// TIA Portal V20 program export: 4 tag tables, 3 data types, 2 data blocks, 7 code blocks (in call order from the OBs), 2 instance data blocks

VAR_GLOBAL   // PLC tag table "Inputs Equipment"
   i_xSabload_Part1_p1_LR AT %I1.0 : Bool;   // Input - Sabload part 1 sensor - table P1 for Left and Right Jig
   i_xSabload_Part2_p1_L AT %I1.1 : Bool;   // Input - Sabload part 2 sensor - table P1 for Left Jig
   i_xSabload_Part3_p1_L AT %I1.2 : Bool;   // Input - Sabload part 3 sensor - table P1 for Left Jig
   i_xSabload_Part4_p1_LR AT %I1.3 : Bool;   // Input - Sabload part 4 sensor - table P1 for Left and Right Jig
   i_xSabload_Part2_p1_R AT %I1.4 : Bool;   // Input - Sabload part 2 sensor - table P1 for Right Jig
   i_xSabload_Part3_p1_R AT %I1.5 : Bool;   // Input - Sabload part 3 sensor - table P1 for Right Jig
   i_xSabload_Part1_p2_LR AT %I1.6 : Bool;   // Input - Sabload part 1 sensor - table P2 for Left and Right Jig
   i_xSabload_Part2_p2_L AT %I1.7 : Bool;   // Input - Sabload part 2 sensor - table P2 for Left Jig
   i_xSabload_Part3_p2_L AT %I2.0 : Bool;   // Input - Sabload part 3 sensor - table P2 for Left Jig
   i_xSabload_Part4_p2_LR AT %I2.1 : Bool;   // Input - Sabload part 4 sensor - table P2 for Left and Right Jig
   i_xSabload_Part2_p2_R AT %I2.2 : Bool;   // Input - Sabload part 2 sensor - table P2 for Right Jig
   i_xSabload_Part3_p2_R AT %I2.3 : Bool;   // Input - Sabload part 3 sensor - table P2 for Right Jig
   i_xBas342_ProgBit0 AT %I0.0 : Bool;   // Input - Bas 342 prog bit 0 for left side Jig
   i_xBas342_ProgBit1 AT %I0.1 : Bool;   // Input - Bas 342 prog bit 1 for Right side Jig
   i_xTableCheck_JigPresent_p1 AT %I0.2 : Bool;   // Input: TableCheck process 1 Sensor for Jig presence for Table P1
   i_xTableCheck_JigPresent_p2 AT %I0.3 : Bool;   // Input: TableCheck process 1 Sensor for Jig presence for Table P2
END_VAR

VAR_GLOBAL   // PLC tag table "OutPut Equipment"
   q_xTableCheck_LampNG_p1 AT %Q5.0 : Bool;   // Output - indication lamp, NO good operation for table P1
   q_xTableCheck_LampOK_p1 AT %Q5.1 : Bool;   // Output - indication lamp, Ok operation for table P1
   q_xTableCheck_LampNG_p2 AT %Q5.2 : Bool;   // Output - indication lamp, NO good operation for table P2
   q_xTableCheck_LampOK_p2 AT %Q5.3 : Bool;   // Output - indication lamp, Ok operation for table P2
END_VAR

VAR_GLOBAL   // PLC tag table "Inputs Machine"
END_VAR

VAR_GLOBAL   // PLC tag table "Output Machine"
END_VAR

TYPE "UDT-BAS342"
VERSION : 0.1
   STRUCT
      Sts : Struct   // Status structure
         xFaulted : Bool;   // wrong program
         xWrongJigProgram : Bool;   // Wrong jig Program by the bus machine
         xNoprogram : Bool;
      END_STRUCT;
      Cmd : Struct   // Command structure
         xCorrectJigProgram : Bool;   // Correct jig Program by the bus machine
         xLeftJig : Bool;   // Bit for the program form the Bas machine
         xRightJig : Bool;   // Bit for the program form the Bas machine
         Spare : Bool;
      END_STRUCT;
      Cfg : Struct   // Configuration structure
         xSpare : Bool;   // Spare
      END_STRUCT;
      Flt : Struct   // Fault structure
         wTrigger : Word;   // Fault triggers
      END_STRUCT;
   END_STRUCT;

END_TYPE

TYPE "UDT-SABload"
VERSION : 0.1
   STRUCT
      Sts : Struct   // Status structure
         axSesnor : Array[1..4] of Bool;
         xCorrectpart : Bool;   // correct part indicaton
         faulted : Bool;   // the module is faulted
         State : Int;   // state machine value
      END_STRUCT;
      Cmd : Struct   // Command structure
         spare : Bool;
      END_STRUCT;
      Cfg : Struct   // Configuration structure
         xSpare : Bool;   // Spare
      END_STRUCT;
      Flt : Struct   // Fault structure
         wTrigger : Word;   // Fault triggers
      END_STRUCT;
   END_STRUCT;

END_TYPE

TYPE "UDT-TableCheck"
VERSION : 0.1
   STRUCT
      Sts : Struct   // Status structure
         xFaulted : Bool;   // System is in faulted state
         xStartSensor : Bool;   // Spare
         xLeftJigplaced : Bool;   // Left Jig is pleased with Left Bas sew program 
         xRightJigPlaced : Bool;   // Right Jig is pleased with Right Bas sew program 
         "xCorrect part" : Bool;   //  the part of the airbage is placed correctly
      END_STRUCT;
      Cmd : Struct   // Command structure
         xJigpresent : Bool;
         spare : Bool;
      END_STRUCT;
      Flt : Struct   // fault structure
         wTrigger : Byte;   // fault trigger word
      END_STRUCT;
   END_STRUCT;

END_TYPE

DATA_BLOCK "DB - Equipment"   // DB4
{ S7_Optimized_Access := 'TRUE' }
// stored: MemoryReserve 100
   VAR
      TableCheckProcess1 : "UDT-TableCheck";
      TableCheckProcess2 : "UDT-TableCheck";
      "SabLaodProcess1-L" { S7_SetPoint := 'True'} : "UDT-SABload";
      "SabLaodProcess1-R" { S7_SetPoint := 'True'} : "UDT-SABload";
      "SabLaodProcess2-L" { S7_SetPoint := 'True'} : "UDT-SABload";
      "SabLaodProcess2-R" { S7_SetPoint := 'True'} : "UDT-SABload";
      Bas342 { S7_SetPoint := 'True'} : "UDT-BAS342";
   END_VAR
BEGIN
END_DATA_BLOCK

DATA_BLOCK "DB - Machine"   // DB3
{ S7_Optimized_Access := 'TRUE' }
// stored: MemoryReserve 100
BEGIN
END_DATA_BLOCK

ORGANIZATION_BLOCK "Main"   // OB1, LAD, ProgramCycle
TITLE = "Main Program Sweep (Cycle)"
{ S7_Optimized_Access := 'TRUE' }
// stored: SetENOAutomatically false
   VAR_INPUT
      Initial_Call : Bool;   // Initial call of this OB
      Remanence : Bool;   // =True, if remanent data are available
   END_VAR
BEGIN

REGION Network 1: CALL - Main machine modules (Not used)
   // Call of the application's main machine functions (NOT used)
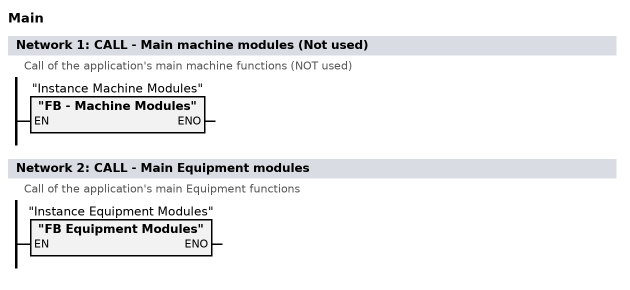
   RUNG wire#powerrail
      "Instance Machine Modules"()
   END_RUNG
   // the same network as SCL:
   "Instance Machine Modules"();   // "FB - Machine Modules"
END_REGION

REGION Network 2: CALL - Main Equipment modules
   // Call of the application's main Equipment functions
   RUNG wire#powerrail
      "Instance Equipment Modules"()
   END_RUNG
   // the same network as SCL:
   "Instance Equipment Modules"();   // "FB Equipment Modules"
END_REGION
END_ORGANIZATION_BLOCK

FUNCTION_BLOCK "FB - Machine Modules"   // FB1, LAD
TITLE = Machine - Modules
{ S7_Optimized_Access := 'TRUE' }
// stored: MemoryReserve 100, SetENOAutomatically false
BEGIN

REGION Network 1: StateHandler process 1 - table
END_REGION

REGION Network 2: StateHandler process 2 - table
END_REGION
END_FUNCTION_BLOCK

FUNCTION_BLOCK "FB Equipment Modules"   // FB2, LAD
TITLE = FB - Equipment Modules
{ S7_Optimized_Access := 'TRUE' }
// stored: MemoryReserve 100, SetENOAutomatically false
   VAR
      "Instance - Bas342" { S7_SetPoint := 'True'} : "FB - Bas342";
      "Instance - TableCheck - Process1" { S7_SetPoint := 'True'} : "FB - TableCheck";
      "Instance - TableCheck - Process2" { S7_SetPoint := 'True'} : "FB - TableCheck";
      "Instance - Sabload - P1 Left" { S7_SetPoint := 'True'} : "FB - Sabload";
      "Instance - Sabload - P1 Right" { S7_SetPoint := 'True'} : "FB - Sabload";
      "Instance - Sabload - P2 Left" { S7_SetPoint := 'True'} : "FB - Sabload";
      "Instance - Sabload - P2 Right" { S7_SetPoint := 'True'} : "FB - Sabload";
   END_VAR
BEGIN

REGION Network 1: Module - Bas342
   // Call of the Bas342 module.
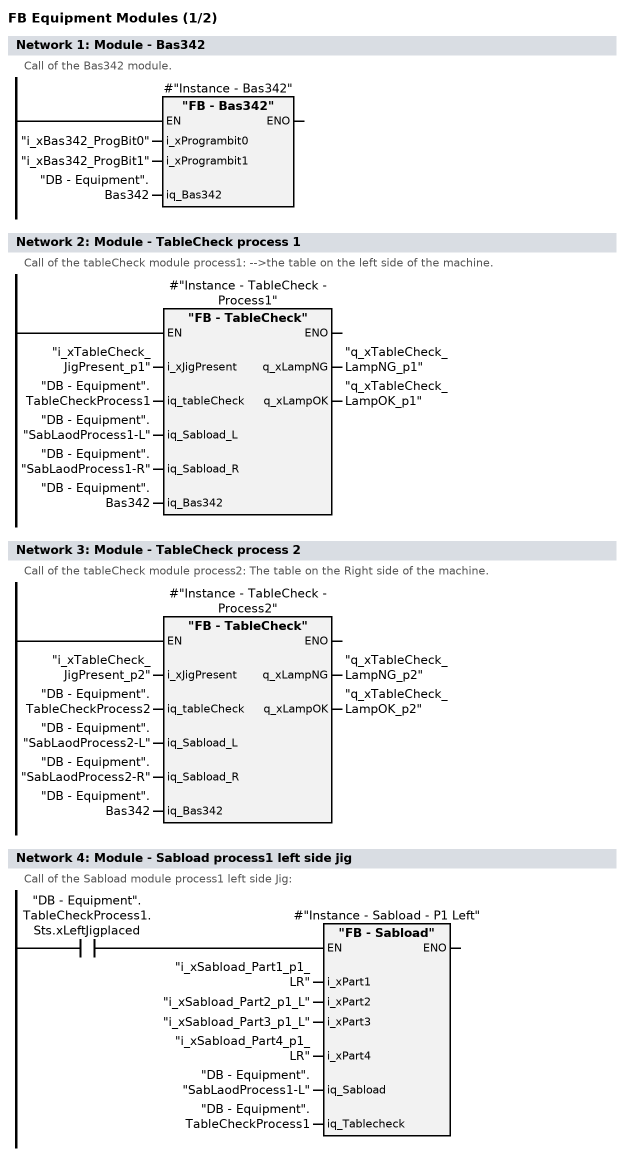
   RUNG wire#powerrail
      #"Instance - Bas342"(i_xProgrambit0 := "i_xBas342_ProgBit0", i_xProgrambit1 := "i_xBas342_ProgBit1", iq_Bas342 := "DB - Equipment".Bas342)
   END_RUNG
   // the same network as SCL:
   #"Instance - Bas342"(i_xProgrambit0 := "i_xBas342_ProgBit0",   // "FB - Bas342"
                        i_xProgrambit1 := "i_xBas342_ProgBit1",
                        iq_Bas342 := "DB - Equipment".Bas342);
END_REGION

REGION Network 2: Module - TableCheck process 1
   // Call of the tableCheck module process1: -->the table on the left side of the machine.
   RUNG wire#powerrail
      #"Instance - TableCheck - Process1"(i_xJigPresent := "i_xTableCheck_JigPresent_p1", iq_tableCheck := "DB - Equipment".TableCheckProcess1, iq_Sabload_L := "DB - Equipment"."SabLaodProcess1-L", iq_Sabload_R := "DB - Equipment"."SabLaodProcess1-R", iq_Bas342 := "DB - Equipment".Bas342, q_xLampNG => "q_xTableCheck_LampNG_p1", q_xLampOK => "q_xTableCheck_LampOK_p1")
   END_RUNG
   // the same network as SCL:
   #"Instance - TableCheck - Process1"(i_xJigPresent := "i_xTableCheck_JigPresent_p1",   // "FB - TableCheck"
                           iq_tableCheck := "DB - Equipment".TableCheckProcess1,
                           iq_Sabload_L := "DB - Equipment"."SabLaodProcess1-L",
                           iq_Sabload_R := "DB - Equipment"."SabLaodProcess1-R",
                           iq_Bas342 := "DB - Equipment".Bas342,
                           q_xLampNG => "q_xTableCheck_LampNG_p1",
                           q_xLampOK => "q_xTableCheck_LampOK_p1");
END_REGION

REGION Network 3: Module - TableCheck process 2
   // Call of the tableCheck module process2: The table on the Right side of the machine.
   RUNG wire#powerrail
      #"Instance - TableCheck - Process2"(i_xJigPresent := "i_xTableCheck_JigPresent_p2", iq_tableCheck := "DB - Equipment".TableCheckProcess2, iq_Sabload_L := "DB - Equipment"."SabLaodProcess2-L", iq_Sabload_R := "DB - Equipment"."SabLaodProcess2-R", iq_Bas342 := "DB - Equipment".Bas342, q_xLampNG => "q_xTableCheck_LampNG_p2", q_xLampOK => "q_xTableCheck_LampOK_p2")
   END_RUNG
   // the same network as SCL:
   #"Instance - TableCheck - Process2"(i_xJigPresent := "i_xTableCheck_JigPresent_p2",   // "FB - TableCheck"
                           iq_tableCheck := "DB - Equipment".TableCheckProcess2,
                           iq_Sabload_L := "DB - Equipment"."SabLaodProcess2-L",
                           iq_Sabload_R := "DB - Equipment"."SabLaodProcess2-R",
                           iq_Bas342 := "DB - Equipment".Bas342,
                           q_xLampNG => "q_xTableCheck_LampNG_p2",
                           q_xLampOK => "q_xTableCheck_LampOK_p2");
END_REGION

REGION Network 4: Module - Sabload process1 left side jig
   // Call of the Sabload module process1 left side Jig:
   RUNG wire#powerrail
      Contact( "DB - Equipment".TableCheckProcess1.Sts.xLeftJigplaced )
      #"Instance - Sabload - P1 Left"(i_xPart1 := "i_xSabload_Part1_p1_LR", i_xPart2 := "i_xSabload_Part2_p1_L", i_xPart3 := "i_xSabload_Part3_p1_L", i_xPart4 := "i_xSabload_Part4_p1_LR", iq_Sabload := "DB - Equipment"."SabLaodProcess1-L", iq_Tablecheck := "DB - Equipment".TableCheckProcess1)
   END_RUNG
   // the same network as SCL:
   IF "DB - Equipment".TableCheckProcess1.Sts.xLeftJigplaced THEN
       #"Instance - Sabload - P1 Left"(i_xPart1 := "i_xSabload_Part1_p1_LR",   // "FB - Sabload"
                               i_xPart2 := "i_xSabload_Part2_p1_L",
                               i_xPart3 := "i_xSabload_Part3_p1_L",
                               i_xPart4 := "i_xSabload_Part4_p1_LR",
                               iq_Sabload := "DB - Equipment"."SabLaodProcess1-L",
                               iq_Tablecheck := "DB - Equipment".TableCheckProcess1);
   END_IF;
END_REGION

REGION Network 5: Module - Sabload process1 Right side jig
   // Call of the Sabload module process1 Right side Jig:
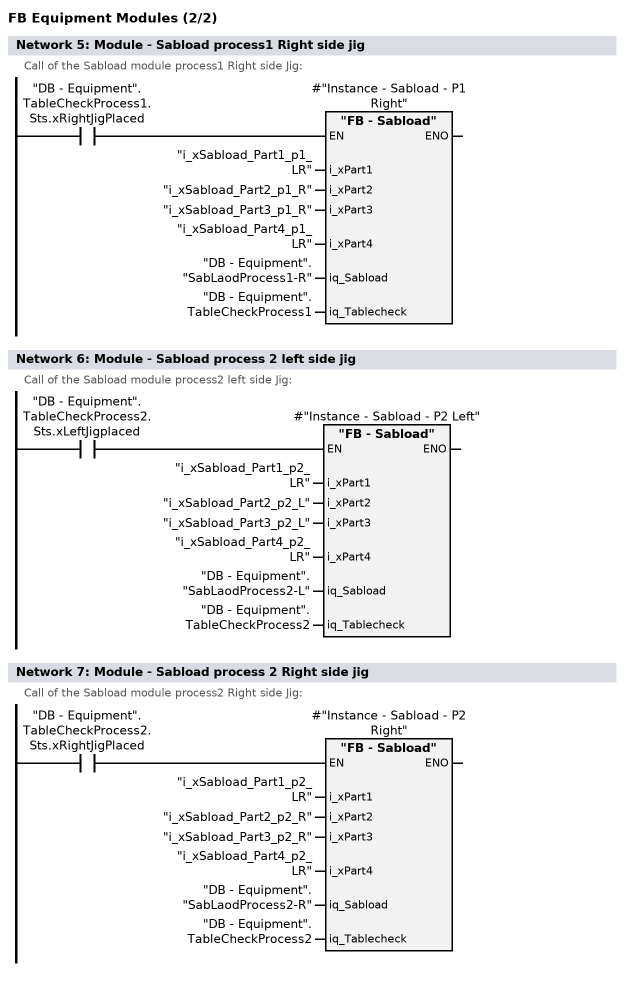
   RUNG wire#powerrail
      Contact( "DB - Equipment".TableCheckProcess1.Sts.xRightJigPlaced )
      #"Instance - Sabload - P1 Right"(i_xPart1 := "i_xSabload_Part1_p1_LR", i_xPart2 := "i_xSabload_Part2_p1_R", i_xPart3 := "i_xSabload_Part3_p1_R", i_xPart4 := "i_xSabload_Part4_p1_LR", iq_Sabload := "DB - Equipment"."SabLaodProcess1-R", iq_Tablecheck := "DB - Equipment".TableCheckProcess1)
   END_RUNG
   // the same network as SCL:
   IF "DB - Equipment".TableCheckProcess1.Sts.xRightJigPlaced THEN
       #"Instance - Sabload - P1 Right"(i_xPart1 := "i_xSabload_Part1_p1_LR",   // "FB - Sabload"
                               i_xPart2 := "i_xSabload_Part2_p1_R",
                               i_xPart3 := "i_xSabload_Part3_p1_R",
                               i_xPart4 := "i_xSabload_Part4_p1_LR",
                               iq_Sabload := "DB - Equipment"."SabLaodProcess1-R",
                               iq_Tablecheck := "DB - Equipment".TableCheckProcess1);
   END_IF;
END_REGION

REGION Network 6: Module - Sabload process 2 left side jig
   // Call of the Sabload module process2 left side Jig:
   RUNG wire#powerrail
      Contact( "DB - Equipment".TableCheckProcess2.Sts.xLeftJigplaced )
      #"Instance - Sabload - P2 Left"(i_xPart1 := "i_xSabload_Part1_p2_LR", i_xPart2 := "i_xSabload_Part2_p2_L", i_xPart3 := "i_xSabload_Part3_p2_L", i_xPart4 := "i_xSabload_Part4_p2_LR", iq_Sabload := "DB - Equipment"."SabLaodProcess2-L", iq_Tablecheck := "DB - Equipment".TableCheckProcess2)
   END_RUNG
   // the same network as SCL:
   IF "DB - Equipment".TableCheckProcess2.Sts.xLeftJigplaced THEN
       #"Instance - Sabload - P2 Left"(i_xPart1 := "i_xSabload_Part1_p2_LR",   // "FB - Sabload"
                               i_xPart2 := "i_xSabload_Part2_p2_L",
                               i_xPart3 := "i_xSabload_Part3_p2_L",
                               i_xPart4 := "i_xSabload_Part4_p2_LR",
                               iq_Sabload := "DB - Equipment"."SabLaodProcess2-L",
                               iq_Tablecheck := "DB - Equipment".TableCheckProcess2);
   END_IF;
END_REGION

REGION Network 7: Module - Sabload process 2 Right side jig
   // Call of the Sabload module process2 Right side Jig:
   RUNG wire#powerrail
      Contact( "DB - Equipment".TableCheckProcess2.Sts.xRightJigPlaced )
      #"Instance - Sabload - P2 Right"(i_xPart1 := "i_xSabload_Part1_p2_LR", i_xPart2 := "i_xSabload_Part2_p2_R", i_xPart3 := "i_xSabload_Part3_p2_R", i_xPart4 := "i_xSabload_Part4_p2_LR", iq_Sabload := "DB - Equipment"."SabLaodProcess2-R", iq_Tablecheck := "DB - Equipment".TableCheckProcess2)
   END_RUNG
   // the same network as SCL:
   IF "DB - Equipment".TableCheckProcess2.Sts.xRightJigPlaced THEN
       #"Instance - Sabload - P2 Right"(i_xPart1 := "i_xSabload_Part1_p2_LR",   // "FB - Sabload"
                               i_xPart2 := "i_xSabload_Part2_p2_R",
                               i_xPart3 := "i_xSabload_Part3_p2_R",
                               i_xPart4 := "i_xSabload_Part4_p2_LR",
                               iq_Sabload := "DB - Equipment"."SabLaodProcess2-R",
                               iq_Tablecheck := "DB - Equipment".TableCheckProcess2);
   END_IF;
END_REGION
END_FUNCTION_BLOCK

FUNCTION_BLOCK "FB - Bas342"   // FB6, LAD
TITLE = Equipment - Bas342
{ S7_Optimized_Access := 'TRUE' }
// This Function blick contain all the logic for controlling a Bas342 module.
// --This module basically for BAS342 sewing machine.
// It is consist of two program bits from BAS342.
// >> Block created by: Engr. Awais Ali
// >> Block creation date:  08-10-2025
// stored: MemoryReserve 100, SetENOAutomatically false
   VAR_INPUT
      i_xProgrambit0 : Bool;
      i_xProgrambit1 : Bool;
   END_VAR
   VAR_IN_OUT
      iq_Bas342 : "UDT-BAS342";
   END_VAR
BEGIN

REGION Network 1: Control - left jig
   // Bit 0 represent the left jig program.
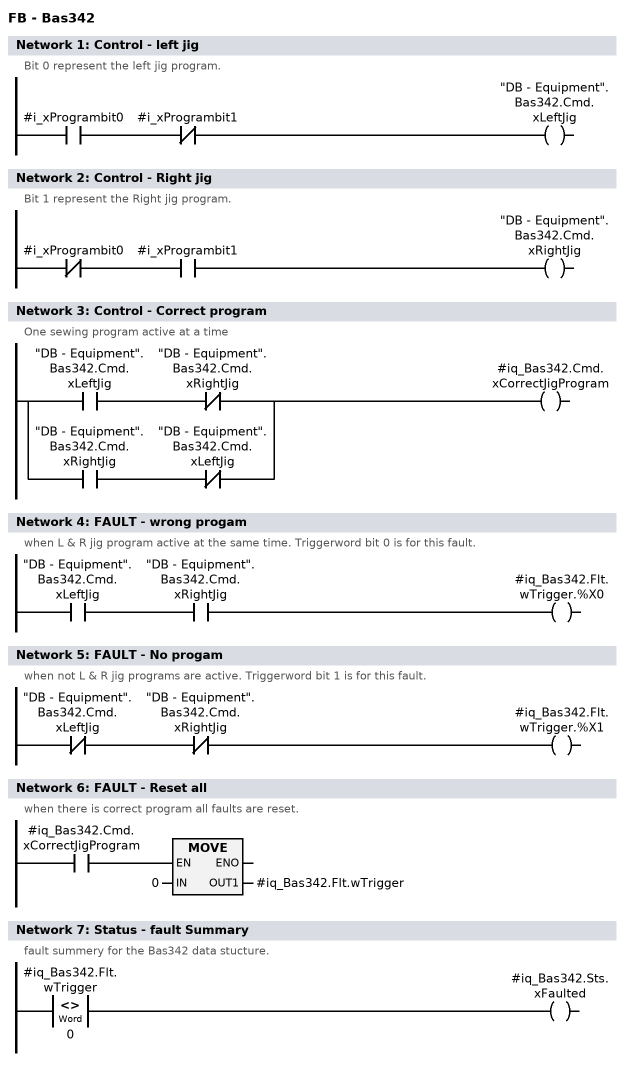
   RUNG wire#powerrail
      Contact( #i_xProgrambit0 )
      I_Contact( #i_xProgrambit1 )
      Coil( "DB - Equipment".Bas342.Cmd.xLeftJig )
   END_RUNG
   // the same network as SCL:
   "DB - Equipment".Bas342.Cmd.xLeftJig := #i_xProgrambit0 AND NOT #i_xProgrambit1;
END_REGION

REGION Network 2: Control - Right jig
   // Bit 1 represent the Right jig program.
   RUNG wire#powerrail
      I_Contact( #i_xProgrambit0 )
      Contact( #i_xProgrambit1 )
      Coil( "DB - Equipment".Bas342.Cmd.xRightJig )
   END_RUNG
   // the same network as SCL:
   "DB - Equipment".Bas342.Cmd.xRightJig := NOT #i_xProgrambit0 AND #i_xProgrambit1;
END_REGION

REGION Network 3: Control - Correct program
   // One sewing program active at a time
   RUNG wire#powerrail
      Contact( "DB - Equipment".Bas342.Cmd.xLeftJig )
      I_Contact( "DB - Equipment".Bas342.Cmd.xRightJig )
      wire#w1
      Coil( #iq_Bas342.Cmd.xCorrectJigProgram )
   END_RUNG
   RUNG wire#powerrail
      Contact( "DB - Equipment".Bas342.Cmd.xRightJig )
      I_Contact( "DB - Equipment".Bas342.Cmd.xLeftJig )
   END_RUNG wire#w1
   // the same network as SCL:
   #iq_Bas342.Cmd.xCorrectJigProgram := ("DB - Equipment".Bas342.Cmd.xLeftJig AND NOT "DB - Equipment".Bas342.Cmd.xRightJig) OR ("DB - Equipment".Bas342.Cmd.xRightJig AND NOT "DB - Equipment".Bas342.Cmd.xLeftJig);
END_REGION

REGION Network 4: FAULT - wrong progam
   // when L & R jig program active at the same time. Triggerword bit 0 is for this fault.
   RUNG wire#powerrail
      Contact( "DB - Equipment".Bas342.Cmd.xLeftJig )
      Contact( "DB - Equipment".Bas342.Cmd.xRightJig )
      Coil( #iq_Bas342.Flt.wTrigger.%X0 )
   END_RUNG
   // the same network as SCL:
   #iq_Bas342.Flt.wTrigger.%X0 := "DB - Equipment".Bas342.Cmd.xLeftJig AND "DB - Equipment".Bas342.Cmd.xRightJig;
END_REGION

REGION Network 5: FAULT - No progam
   // when not L & R jig programs are active. Triggerword bit 1 is for this fault.
   RUNG wire#powerrail
      I_Contact( "DB - Equipment".Bas342.Cmd.xLeftJig )
      I_Contact( "DB - Equipment".Bas342.Cmd.xRightJig )
      Coil( #iq_Bas342.Flt.wTrigger.%X1 )
   END_RUNG
   // the same network as SCL:
   #iq_Bas342.Flt.wTrigger.%X1 := NOT "DB - Equipment".Bas342.Cmd.xLeftJig AND NOT "DB - Equipment".Bas342.Cmd.xRightJig;
END_REGION

REGION Network 6: FAULT - Reset all
   // when there is correct program all faults are reset.
   RUNG wire#powerrail
      Contact( #iq_Bas342.Cmd.xCorrectJigProgram )
      Move(in := 0, out1 => #iq_Bas342.Flt.wTrigger)
   END_RUNG
   // the same network as SCL:
   IF #iq_Bas342.Cmd.xCorrectJigProgram THEN #iq_Bas342.Flt.wTrigger := 0; END_IF;
END_REGION

REGION Network 7: Status - fault Summary
   // fault summery for the Bas342 data stucture.
   RUNG wire#powerrail
      { S7_Templates := "SrcType := Word" } NE_Contact(in1 := #iq_Bas342.Flt.wTrigger, in2 := 0)
      Coil( #iq_Bas342.Sts.xFaulted )
   END_RUNG
   // the same network as SCL:
   #iq_Bas342.Sts.xFaulted := #iq_Bas342.Flt.wTrigger <> 0;
END_REGION
END_FUNCTION_BLOCK

FUNCTION_BLOCK "FB - TableCheck"   // FB3, LAD
TITLE = Equipment - TableCheck
{ S7_Optimized_Access := 'TRUE' }
// This function block contains all logic for controlling a TableCheck module.
// -This module consists of a table, a jig presense sensor and Indication lamp Red (NG) and green (Ok).
// 
// >> Block created by: Engr. Awais Ali
// >> Block creation date:  08-10-2025
// stored: MemoryReserve 100, SetENOAutomatically false
   VAR_INPUT
      i_xJigPresent : Bool;
   END_VAR
   VAR_OUTPUT
      q_xLampNG : Bool;
      q_xLampOK : Bool;
   END_VAR
   VAR_IN_OUT
      iq_tableCheck : "UDT-TableCheck";
      iq_Sabload_L : "UDT-SABload";
      iq_Sabload_R : "UDT-SABload";
      iq_Bas342 : "UDT-BAS342";
   END_VAR
   VAR
      iState : Int;
      OnDelay_JigL { S7_SetPoint := 'True'} : TON_TIME;
      OffDelay_JigL { S7_SetPoint := 'True'} : TOF_TIME;
      OnDelay_JigR { S7_SetPoint := 'True'} : TON_TIME;
      OffDelay_JigR { S7_SetPoint := 'True'} : TOF_TIME;
   END_VAR
BEGIN

REGION Network 1: control - left jig
   // Detect the presence of left side Jig.
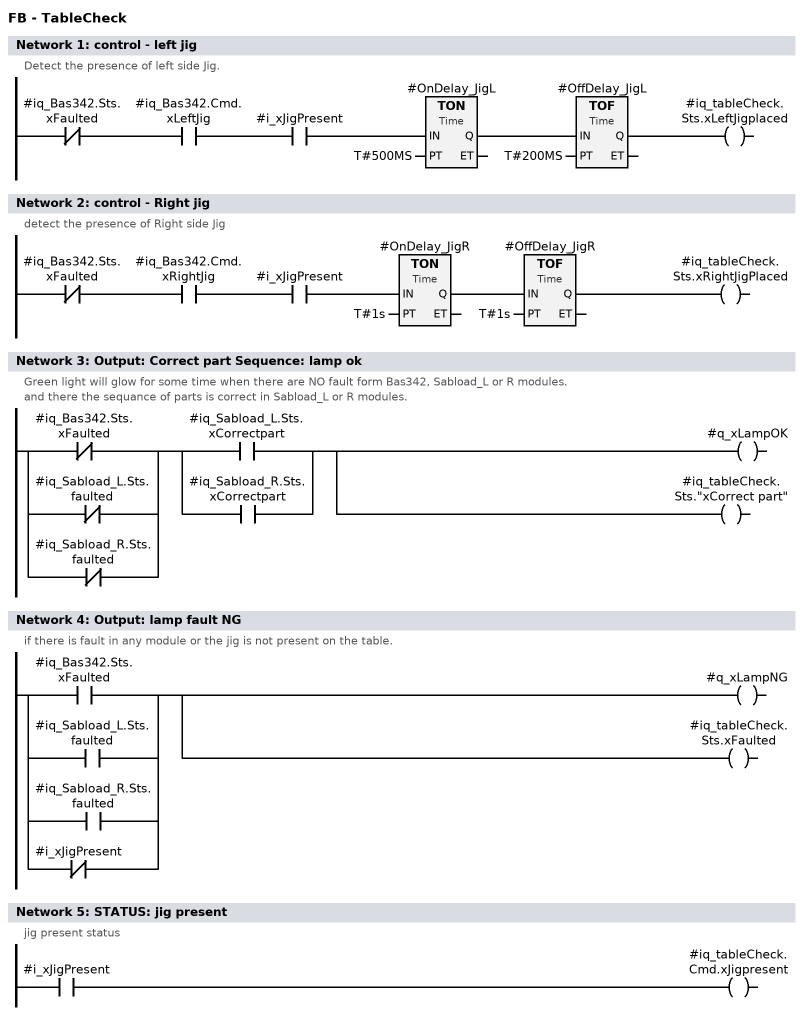
   RUNG wire#powerrail
      I_Contact( #iq_Bas342.Sts.xFaulted )
      Contact( #iq_Bas342.Cmd.xLeftJig )
      Contact( #i_xJigPresent )
      { S7_Templates := "time_type := Time" } #OnDelay_JigL.TON(pt := T#500MS, et =>)
      { S7_Templates := "time_type := Time" } #OffDelay_JigL.TOF(pt := T#200MS, et =>)
      Coil( #iq_tableCheck.Sts.xLeftJigplaced )
   END_RUNG
   // the same network as SCL:
   #OnDelay_JigL(IN := NOT #iq_Bas342.Sts.xFaulted AND #iq_Bas342.Cmd.xLeftJig AND #i_xJigPresent,   // TON
                 PT := T#500MS);
   #OffDelay_JigL(IN := #OnDelay_JigL.Q, PT := T#200MS);   // TOF
   #iq_tableCheck.Sts.xLeftJigplaced := #OffDelay_JigL.Q;
END_REGION

REGION Network 2: control - Right jig
   // detect the presence of Right side Jig
   RUNG wire#powerrail
      I_Contact( #iq_Bas342.Sts.xFaulted )
      Contact( #iq_Bas342.Cmd.xRightJig )
      Contact( #i_xJigPresent )
      { S7_Templates := "time_type := Time" } #OnDelay_JigR.TON(pt := T#1s, et =>)
      { S7_Templates := "time_type := Time" } #OffDelay_JigR.TOF(pt := T#1s, et =>)
      Coil( #iq_tableCheck.Sts.xRightJigPlaced )
   END_RUNG
   // the same network as SCL:
   #OnDelay_JigR(IN := NOT #iq_Bas342.Sts.xFaulted AND #iq_Bas342.Cmd.xRightJig AND #i_xJigPresent, PT := T#1s);   // TON
   #OffDelay_JigR(IN := #OnDelay_JigR.Q, PT := T#1s);   // TOF
   #iq_tableCheck.Sts.xRightJigPlaced := #OffDelay_JigR.Q;
END_REGION

REGION Network 3: Output: Correct part Sequence: lamp ok
   // Green light will glow for some time when there are NO fault form Bas342, Sabload_L or R modules. 
   // 
   // and there the sequance of parts is correct in Sabload_L or R modules.
   RUNG wire#powerrail
      I_Contact( #iq_Bas342.Sts.xFaulted )
      wire#w1
      Contact( #iq_Sabload_L.Sts.xCorrectpart )
      wire#w2
      Coil( #q_xLampOK )
   END_RUNG
   RUNG wire#powerrail
      I_Contact( #iq_Sabload_L.Sts.faulted )
   END_RUNG wire#w1
   RUNG wire#powerrail
      I_Contact( #iq_Sabload_R.Sts.faulted )
   END_RUNG wire#w1
   RUNG wire#w1
      Contact( #iq_Sabload_R.Sts.xCorrectpart )
   END_RUNG wire#w2
   RUNG wire#w2
      Coil( #iq_tableCheck.Sts."xCorrect part" )
   END_RUNG
   // the same network as SCL:
   #q_xLampOK := (NOT #iq_Bas342.Sts.xFaulted OR NOT #iq_Sabload_L.Sts.faulted OR NOT #iq_Sabload_R.Sts.faulted) AND (#iq_Sabload_L.Sts.xCorrectpart OR #iq_Sabload_R.Sts.xCorrectpart);
   #iq_tableCheck.Sts."xCorrect part" := #q_xLampOK;
END_REGION

REGION Network 4: Output: lamp fault NG
   // if there is fault in any module or the jig is not present on the table.
   RUNG wire#powerrail
      Contact( #iq_Bas342.Sts.xFaulted )
      wire#w1
      Coil( #q_xLampNG )
   END_RUNG
   RUNG wire#powerrail
      Contact( #iq_Sabload_L.Sts.faulted )
   END_RUNG wire#w1
   RUNG wire#powerrail
      Contact( #iq_Sabload_R.Sts.faulted )
   END_RUNG wire#w1
   RUNG wire#powerrail
      I_Contact( #i_xJigPresent )
   END_RUNG wire#w1
   RUNG wire#w1
      Coil( #iq_tableCheck.Sts.xFaulted )
   END_RUNG
   // the same network as SCL:
   #q_xLampNG := #iq_Bas342.Sts.xFaulted OR #iq_Sabload_L.Sts.faulted OR #iq_Sabload_R.Sts.faulted OR NOT #i_xJigPresent;
   #iq_tableCheck.Sts.xFaulted := #q_xLampNG;
END_REGION

REGION Network 5: STATUS: jig present
   // jig present status
   RUNG wire#powerrail
      Contact( #i_xJigPresent )
      Coil( #iq_tableCheck.Cmd.xJigpresent )
   END_RUNG
   // the same network as SCL:
   #iq_tableCheck.Cmd.xJigpresent := #i_xJigPresent;
END_REGION
END_FUNCTION_BLOCK

FUNCTION_BLOCK "FB - Sabload"   // FB5, LAD
TITLE = Equipment - Sabload
{ S7_Optimized_Access := 'TRUE' }
// This function block contains all logic for controlling a Sabload module.
// -This module consists of a jig, table, airbag part detection layser sensors.
// 
// >> Block created by: Engr. Awais Ali
// >> Block creation date:  08-10-2025
// stored: MemoryReserve 100, SetENOAutomatically false
   VAR_INPUT
      i_xPart1 : Bool;
      i_xPart2 : Bool;
      i_xPart3 : Bool;
      i_xPart4 : Bool;
   END_VAR
   VAR_IN_OUT
      iq_Sabload : "UDT-SABload";
      iq_Tablecheck : "UDT-TableCheck";
   END_VAR
   VAR
      iState : Int;
      OndelayJigPresent { S7_SetPoint := 'True'} : TON_TIME;
      OnDelayPart1 { S7_SetPoint := 'True'} : TON_TIME;
      OnDelayPart2 { S7_SetPoint := 'True'} : TON_TIME;
      OnDelayPart3 { S7_SetPoint := 'True'} : TON_TIME;
      OnDelayPart4 { S7_SetPoint := 'True'} : TON_TIME;
      TriggerS1 : Bool;
      OnDelayReset { S7_SetPoint := 'True'} : TON_TIME;
      TriggerS6 : Bool;
      TriggerS2 { ExternalAccessible := 'False'; ExternalVisible := 'False'; ExternalWritable := 'False'} : Bool;
      TriggerS3 { ExternalAccessible := 'False'; ExternalVisible := 'False'; ExternalWritable := 'False'} : Bool;
      TriggerS4 { ExternalAccessible := 'False'; ExternalVisible := 'False'; ExternalWritable := 'False'} : Bool;
      TriggerS5 { ExternalAccessible := 'False'; ExternalVisible := 'False'; ExternalWritable := 'False'} : Bool;
      Oneshot_IndicationLamp { S7_SetPoint := 'True'} : TP_TIME;
      OnDelay_fault1 { S7_SetPoint := 'True'} : TON_TIME;
      OnDelayPart5 { S7_SetPoint := 'True'} : TON_TIME;
      InstanceTrigger_part1 { S7_SetPoint := 'True'} : R_TRIG;
      InstanceTrigger_part2 { S7_SetPoint := 'True'} : R_TRIG;
      InstanceTrigger_part3 { S7_SetPoint := 'True'} : R_TRIG;
      InstanceTrigger_part4 { S7_SetPoint := 'True'} : R_TRIG;
      xOkPart : Bool;
      xpartOrderComplete : Bool;
      Instance_F_trigger_part1 { S7_SetPoint := 'True'} : F_TRIG;
   END_VAR
   VAR_TEMP   // added for the SCL form of the ladder/FBD networks
      _w1 : Bool;
   END_VAR
BEGIN

REGION Network 1: Control - part one
   // if the 1st part place on the Jig for x seconds the state move from 0 to 5. It confirm the part is there.
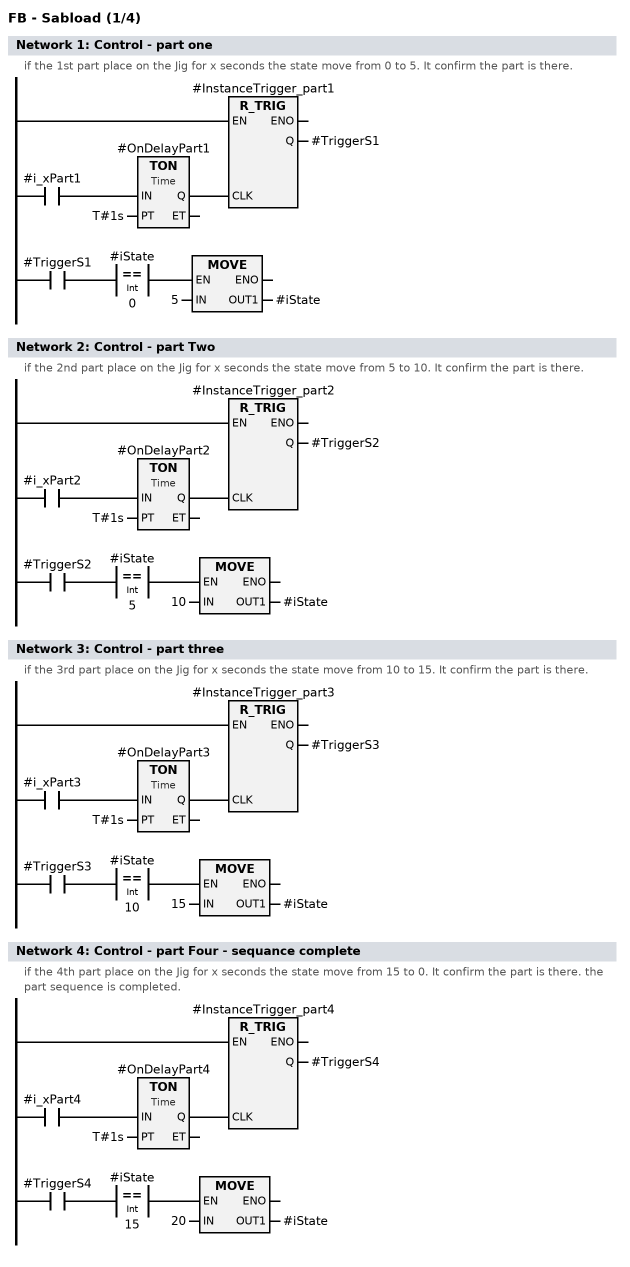
   RUNG wire#powerrail
      #InstanceTrigger_part1.R_TRIG(CLK := wire#w1, Q => #TriggerS1)
   END_RUNG
   RUNG wire#powerrail
      Contact( #i_xPart1 )
      { S7_Templates := "time_type := Time" } #OnDelayPart1.TON(pt := T#1s, et =>)
   END_RUNG wire#w1
   RUNG wire#powerrail
      Contact( #TriggerS1 )
      { S7_Templates := "SrcType := Int" } EQ_Contact(in1 := #iState, in2 := 0)
      Move(in := 5, out1 => #iState)
   END_RUNG
   // the same network as SCL:
   #OnDelayPart1(IN := #i_xPart1, PT := T#1s);   // TON
   #InstanceTrigger_part1(CLK := #OnDelayPart1.Q, Q => #TriggerS1);   // R_TRIG
   IF #TriggerS1 AND (#iState = 0) THEN #iState := 5; END_IF;
END_REGION

REGION Network 2: Control - part Two
   // if the 2nd part place on the Jig for x seconds the state move from 5 to 10. It confirm the part is there.
   RUNG wire#powerrail
      #InstanceTrigger_part2.R_TRIG(CLK := wire#w1, Q => #TriggerS2)
   END_RUNG
   RUNG wire#powerrail
      Contact( #i_xPart2 )
      { S7_Templates := "time_type := Time" } #OnDelayPart2.TON(pt := T#1s, et =>)
   END_RUNG wire#w1
   RUNG wire#powerrail
      Contact( #TriggerS2 )
      { S7_Templates := "SrcType := Int" } EQ_Contact(in1 := #iState, in2 := 5)
      Move(in := 10, out1 => #iState)
   END_RUNG
   // the same network as SCL:
   #OnDelayPart2(IN := #i_xPart2, PT := T#1s);   // TON
   #InstanceTrigger_part2(CLK := #OnDelayPart2.Q, Q => #TriggerS2);   // R_TRIG
   IF #TriggerS2 AND (#iState = 5) THEN #iState := 10; END_IF;
END_REGION

REGION Network 3: Control - part three
   // if the 3rd part place on the Jig for x seconds the state move from 10 to 15. It confirm the part is there.
   RUNG wire#powerrail
      #InstanceTrigger_part3.R_TRIG(CLK := wire#w1, Q => #TriggerS3)
   END_RUNG
   RUNG wire#powerrail
      Contact( #i_xPart3 )
      { S7_Templates := "time_type := Time" } #OnDelayPart3.TON(pt := T#1s, et =>)
   END_RUNG wire#w1
   RUNG wire#powerrail
      Contact( #TriggerS3 )
      { S7_Templates := "SrcType := Int" } EQ_Contact(in1 := #iState, in2 := 10)
      Move(in := 15, out1 => #iState)
   END_RUNG
   // the same network as SCL:
   #OnDelayPart3(IN := #i_xPart3, PT := T#1s);   // TON
   #InstanceTrigger_part3(CLK := #OnDelayPart3.Q, Q => #TriggerS3);   // R_TRIG
   IF #TriggerS3 AND (#iState = 10) THEN #iState := 15; END_IF;
END_REGION

REGION Network 4: Control - part Four - sequance complete
   // if the 4th part place on the Jig for x seconds the state move from 15 to 0. It confirm the part is there. the part sequence is completed.
   RUNG wire#powerrail
      #InstanceTrigger_part4.R_TRIG(CLK := wire#w1, Q => #TriggerS4)
   END_RUNG
   RUNG wire#powerrail
      Contact( #i_xPart4 )
      { S7_Templates := "time_type := Time" } #OnDelayPart4.TON(pt := T#1s, et =>)
   END_RUNG wire#w1
   RUNG wire#powerrail
      Contact( #TriggerS4 )
      { S7_Templates := "SrcType := Int" } EQ_Contact(in1 := #iState, in2 := 15)
      Move(in := 20, out1 => #iState)
   END_RUNG
   // the same network as SCL:
   #OnDelayPart4(IN := #i_xPart4, PT := T#1s);   // TON
   #InstanceTrigger_part4(CLK := #OnDelayPart4.Q, Q => #TriggerS4);   // R_TRIG
   IF #TriggerS4 AND (#iState = 15) THEN #iState := 20; END_IF;
END_REGION

REGION Network 5: Control - Remove the jig: sequance complete
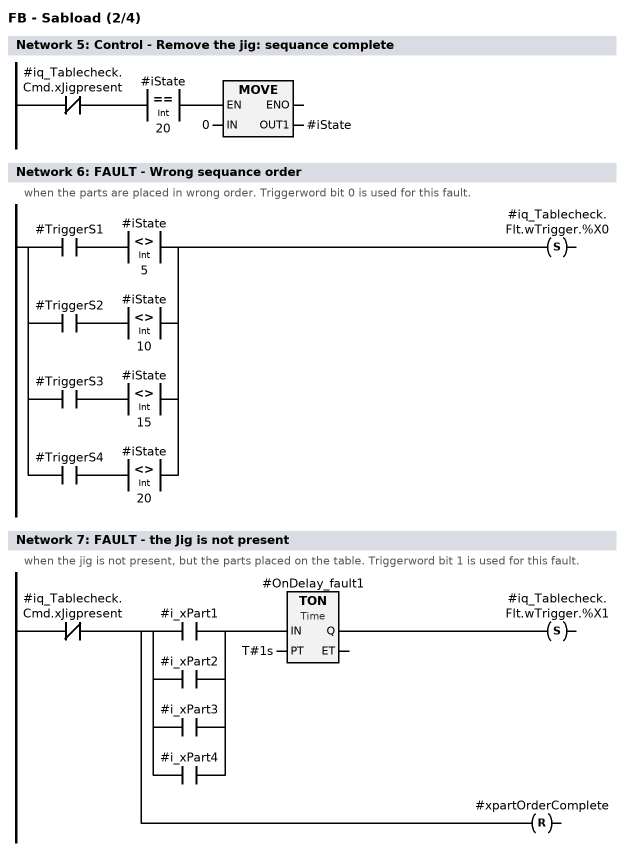
   RUNG wire#powerrail
      I_Contact( #iq_Tablecheck.Cmd.xJigpresent )
      { S7_Templates := "SrcType := Int" } EQ_Contact(in1 := #iState, in2 := 20)
      Move(in := 0, out1 => #iState)
   END_RUNG
   // the same network as SCL:
   IF NOT #iq_Tablecheck.Cmd.xJigpresent AND (#iState = 20) THEN #iState := 0; END_IF;
END_REGION

REGION Network 6: FAULT - Wrong sequance order
   // when the parts are placed in wrong order. Triggerword bit 0 is used for this fault.
   RUNG wire#powerrail
      Contact( #TriggerS1 )
      { S7_Templates := "SrcType := Int" } NE_Contact(in1 := #iState, in2 := 5)
      wire#w1
      S_Coil( #iq_Tablecheck.Flt.wTrigger.%X0 )
   END_RUNG
   RUNG wire#powerrail
      Contact( #TriggerS2 )
      { S7_Templates := "SrcType := Int" } NE_Contact(in1 := #iState, in2 := 10)
   END_RUNG wire#w1
   RUNG wire#powerrail
      Contact( #TriggerS3 )
      { S7_Templates := "SrcType := Int" } NE_Contact(in1 := #iState, in2 := 15)
   END_RUNG wire#w1
   RUNG wire#powerrail
      Contact( #TriggerS4 )
      { S7_Templates := "SrcType := Int" } NE_Contact(in1 := #iState, in2 := 20)
   END_RUNG wire#w1
   // the same network as SCL:
   IF (#TriggerS1 AND (#iState <> 5)) OR (#TriggerS2 AND (#iState <> 10)) OR (#TriggerS3 AND (#iState <> 15)) OR (#TriggerS4 AND (#iState <> 20)) THEN
       #iq_Tablecheck.Flt.wTrigger.%X0 := TRUE;
   END_IF;
END_REGION

REGION Network 7: FAULT - the Jig is not present
   // when the jig is not present, but the parts placed on the table. Triggerword bit 1 is used for this fault.
   RUNG wire#powerrail
      I_Contact( #iq_Tablecheck.Cmd.xJigpresent )
      wire#w1
      Contact( #i_xPart1 )
      wire#w2
      { S7_Templates := "time_type := Time" } #OnDelay_fault1.TON(pt := T#1s, et =>)
      S_Coil( #iq_Tablecheck.Flt.wTrigger.%X1 )
   END_RUNG
   RUNG wire#w1
      Contact( #i_xPart2 )
   END_RUNG wire#w2
   RUNG wire#w1
      Contact( #i_xPart3 )
   END_RUNG wire#w2
   RUNG wire#w1
      Contact( #i_xPart4 )
   END_RUNG wire#w2
   RUNG wire#w1
      R_Coil( #xpartOrderComplete )
   END_RUNG
   // the same network as SCL:
   #_w1 := NOT #iq_Tablecheck.Cmd.xJigpresent;
   #OnDelay_fault1(IN := #_w1 AND (#i_xPart1 OR #i_xPart2 OR #i_xPart3 OR #i_xPart4), PT := T#1s);   // TON
   IF #OnDelay_fault1.Q THEN #iq_Tablecheck.Flt.wTrigger.%X1 := TRUE; END_IF;
   IF #_w1 THEN #xpartOrderComplete := FALSE; END_IF;
END_REGION

REGION Network 8: FAULT - previous parts missing
   // when the palced parts removed before completing the sequnace. Triggerword bit 1 is used for this fault.
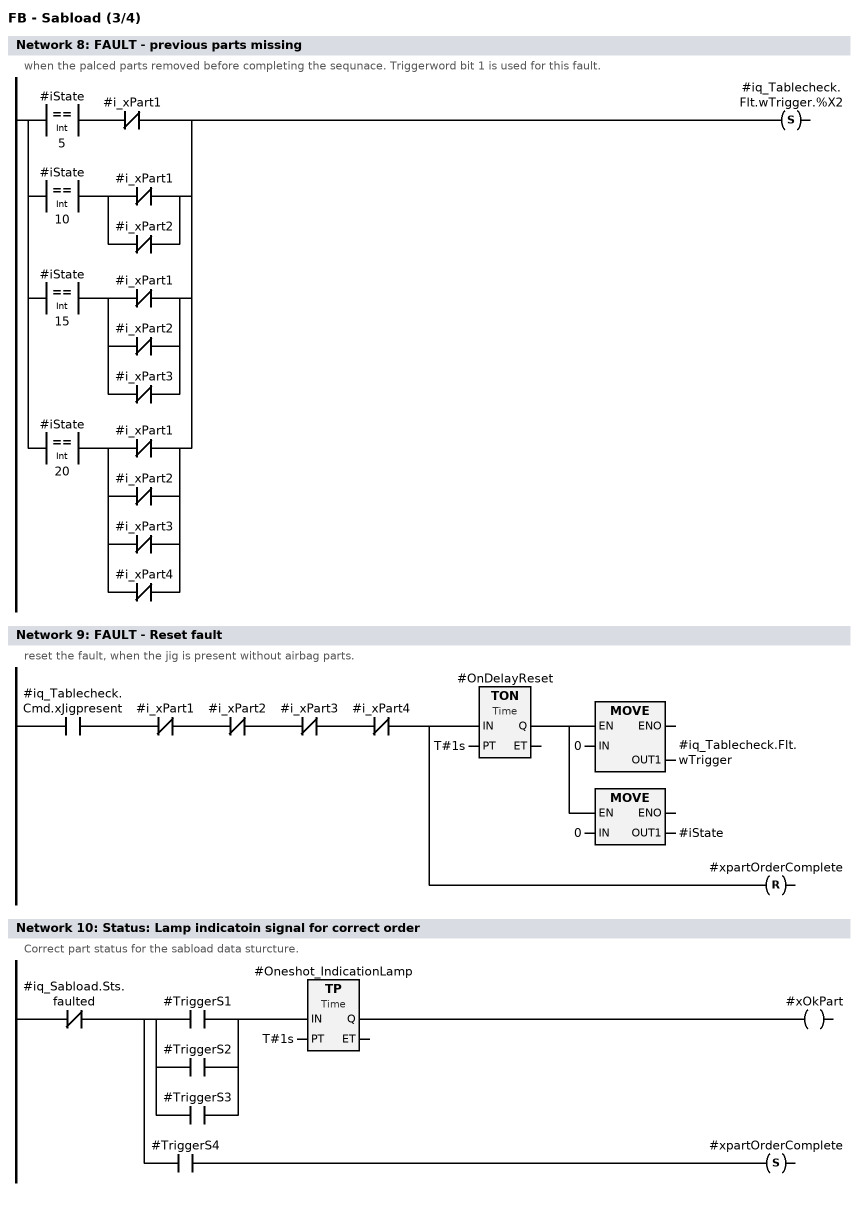
   RUNG wire#powerrail
      { S7_Templates := "SrcType := Int" } EQ_Contact(in1 := #iState, in2 := 5)
      I_Contact( #i_xPart1 )
      wire#w1
      S_Coil( #iq_Tablecheck.Flt.wTrigger.%X2 )
   END_RUNG
   RUNG wire#powerrail
      { S7_Templates := "SrcType := Int" } EQ_Contact(in1 := #iState, in2 := 10)
      wire#w2
      I_Contact( #i_xPart1 )
   END_RUNG wire#w1
   RUNG wire#w2
      I_Contact( #i_xPart2 )
   END_RUNG wire#w1
   RUNG wire#powerrail
      { S7_Templates := "SrcType := Int" } EQ_Contact(in1 := #iState, in2 := 15)
      wire#w3
      I_Contact( #i_xPart1 )
   END_RUNG wire#w1
   RUNG wire#w3
      I_Contact( #i_xPart2 )
   END_RUNG wire#w1
   RUNG wire#w3
      I_Contact( #i_xPart3 )
   END_RUNG wire#w1
   RUNG wire#powerrail
      { S7_Templates := "SrcType := Int" } EQ_Contact(in1 := #iState, in2 := 20)
      wire#w4
      I_Contact( #i_xPart1 )
   END_RUNG wire#w1
   RUNG wire#w4
      I_Contact( #i_xPart2 )
   END_RUNG wire#w1
   RUNG wire#w4
      I_Contact( #i_xPart3 )
   END_RUNG wire#w1
   RUNG wire#w4
      I_Contact( #i_xPart4 )
   END_RUNG wire#w1
   // the same network as SCL:
   IF ((#iState = 5) AND NOT #i_xPart1) OR ((#iState = 10) AND (NOT #i_xPart1 OR NOT #i_xPart2)) OR ((#iState = 15) AND (NOT #i_xPart1 OR NOT #i_xPart2 OR NOT #i_xPart3)) OR ((#iState = 20) AND (NOT #i_xPart1 OR NOT #i_xPart2 OR NOT #i_xPart3 OR NOT #i_xPart4)) THEN
       #iq_Tablecheck.Flt.wTrigger.%X2 := TRUE;
   END_IF;
END_REGION

REGION Network 9: FAULT - Reset fault
   // reset the fault, when the jig is present without airbag parts.
   RUNG wire#powerrail
      Contact( #iq_Tablecheck.Cmd.xJigpresent )
      I_Contact( #i_xPart1 )
      I_Contact( #i_xPart2 )
      I_Contact( #i_xPart3 )
      I_Contact( #i_xPart4 )
      wire#w1
      { S7_Templates := "time_type := Time" } #OnDelayReset.TON(pt := T#1s, et =>)
      wire#w2
      Move(in := 0, out1 => #iq_Tablecheck.Flt.wTrigger)
   END_RUNG
   RUNG wire#w2
      Move(in := 0, out1 => #iState)
   END_RUNG
   RUNG wire#w1
      R_Coil( #xpartOrderComplete )
   END_RUNG
   // the same network as SCL:
   #_w1 := #iq_Tablecheck.Cmd.xJigpresent AND NOT #i_xPart1 AND NOT #i_xPart2 AND NOT #i_xPart3 AND NOT #i_xPart4;
   #OnDelayReset(IN := #_w1, PT := T#1s);   // TON
   IF #OnDelayReset.Q THEN
       #iq_Tablecheck.Flt.wTrigger := 0;
       #iState := 0;
   END_IF;
   IF #_w1 THEN #xpartOrderComplete := FALSE; END_IF;
END_REGION

REGION Network 10: Status: Lamp indicatoin signal for correct order
   // Correct part status for the sabload data sturcture.
   RUNG wire#powerrail
      I_Contact( #iq_Sabload.Sts.faulted )
      wire#w1
      Contact( #TriggerS1 )
      wire#w2
      { S7_Templates := "time_type := Time" } #Oneshot_IndicationLamp.TP(pt := T#1s, et =>)
      Coil( #xOkPart )
   END_RUNG
   RUNG wire#w1
      Contact( #TriggerS2 )
   END_RUNG wire#w2
   RUNG wire#w1
      Contact( #TriggerS3 )
   END_RUNG wire#w2
   RUNG wire#w1
      Contact( #TriggerS4 )
      S_Coil( #xpartOrderComplete )
   END_RUNG
   // the same network as SCL:
   #_w1 := NOT #iq_Sabload.Sts.faulted;
   #Oneshot_IndicationLamp(IN := #_w1 AND (#TriggerS1 OR #TriggerS2 OR #TriggerS3), PT := T#1s);   // TP
   #xOkPart := #Oneshot_IndicationLamp.Q;
   IF #_w1 AND #TriggerS4 THEN #xpartOrderComplete := TRUE; END_IF;
END_REGION

REGION Network 11: the part of the airbage is placed correctly
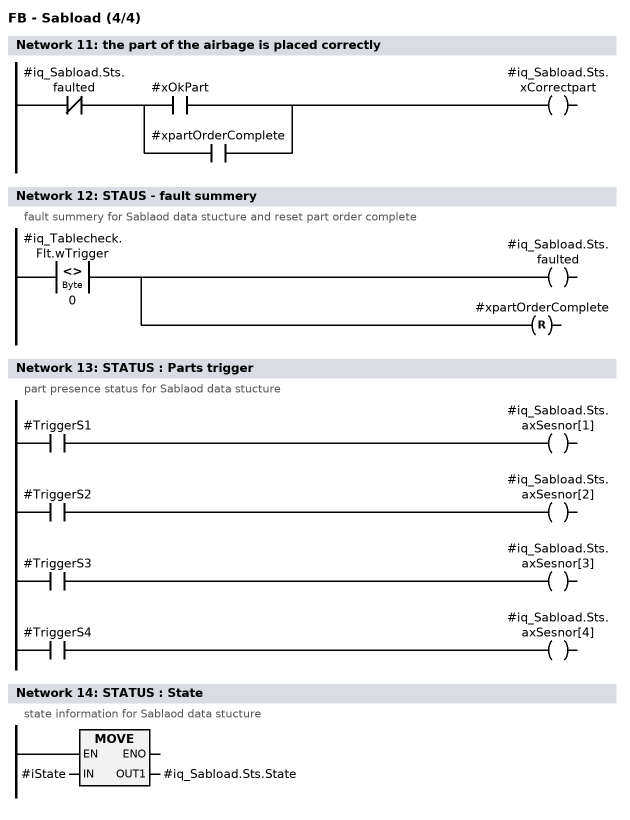
   RUNG wire#powerrail
      I_Contact( #iq_Sabload.Sts.faulted )
      wire#w1
      Contact( #xOkPart )
      wire#w2
      Coil( #iq_Sabload.Sts.xCorrectpart )
   END_RUNG
   RUNG wire#w1
      Contact( #xpartOrderComplete )
   END_RUNG wire#w2
   // the same network as SCL:
   #iq_Sabload.Sts.xCorrectpart := NOT #iq_Sabload.Sts.faulted AND (#xOkPart OR #xpartOrderComplete);
END_REGION

REGION Network 12: STAUS - fault summery
   // fault summery for Sablaod data stucture and reset part order complete
   RUNG wire#powerrail
      { S7_Templates := "SrcType := Byte" } NE_Contact(in1 := #iq_Tablecheck.Flt.wTrigger, in2 := 0)
      wire#w1
      Coil( #iq_Sabload.Sts.faulted )
   END_RUNG
   RUNG wire#w1
      R_Coil( #xpartOrderComplete )
   END_RUNG
   // the same network as SCL:
   #iq_Sabload.Sts.faulted := #iq_Tablecheck.Flt.wTrigger <> 0;
   IF #iq_Sabload.Sts.faulted THEN #xpartOrderComplete := FALSE; END_IF;
END_REGION

REGION Network 13: STATUS : Parts trigger
   // part presence status for Sablaod data stucture
   RUNG wire#powerrail
      Contact( #TriggerS1 )
      Coil( #iq_Sabload.Sts.axSesnor[1] )
   END_RUNG
   RUNG wire#powerrail
      Contact( #TriggerS2 )
      Coil( #iq_Sabload.Sts.axSesnor[2] )
   END_RUNG
   RUNG wire#powerrail
      Contact( #TriggerS3 )
      Coil( #iq_Sabload.Sts.axSesnor[3] )
   END_RUNG
   RUNG wire#powerrail
      Contact( #TriggerS4 )
      Coil( #iq_Sabload.Sts.axSesnor[4] )
   END_RUNG
   // the same network as SCL:
   #iq_Sabload.Sts.axSesnor[1] := #TriggerS1;
   #iq_Sabload.Sts.axSesnor[2] := #TriggerS2;
   #iq_Sabload.Sts.axSesnor[3] := #TriggerS3;
   #iq_Sabload.Sts.axSesnor[4] := #TriggerS4;
END_REGION

REGION Network 14: STATUS : State
   // state information for Sablaod data stucture
   RUNG wire#powerrail
      Move(in := #iState, out1 => #iq_Sabload.Sts.State)
   END_RUNG
   // the same network as SCL:
   #iq_Sabload.Sts.State := #iState;
END_REGION
END_FUNCTION_BLOCK

FUNCTION_BLOCK "FB-counter"
{ S7_Optimized_Access := 'TRUE' }
VERSION : 0.1
   VAR 
      Timer2s {InstructionName := 'TON_TIME'; LibVersion := '1.0'; S7_SetPoint := 'False'} : TON_TIME;
      "Counter" { S7_SetPoint := 'True'} : Int;
   END_VAR


BEGIN
	//ksjadgfksjdflksadf
	////ksjadgfksjdflksadf
	////ksjadgfksjdflksadf
	////ksjadgfksjdflksadf
END_FUNCTION_BLOCK

DATA_BLOCK "Instance Machine Modules"   // DB1
// stored: InstanceOfName FB - Machine Modules, InstanceOfType FB
"FB - Machine Modules"
BEGIN
END_DATA_BLOCK

DATA_BLOCK "Instance Equipment Modules"   // DB2
// stored: InstanceOfName FB Equipment Modules, InstanceOfType FB
"FB Equipment Modules"
BEGIN
END_DATA_BLOCK
